Universal Robots PolyScope program: assembly_app.urp

Program assembly_app (installation=default directory=/home/ur/ursim-current/programs createdIn=5.17.1 lastSavedIn=5.17.1 robotSerialNumber=20195299999)
Calibrated DH parameters: a=[0, -0.6127, -0.57155, 0, 0, 0]; d=[0.1807, 0, 0, 0.17415, 0.11985, 0.11655]; alpha=[1.570796, 0, 0, 1.570796, -1.570796, 0]; deltaTheta=[0, 0, 0, 0, 0, 0]
InitVariablesNode
BeforeStart
  Script file /home/ur/ursim-current/programs/assemby_script_demo.script
    | # HMI input variables
    | approach = 100
    | contact_pose = p[-0.190, -0.610, 0.061, -0.00, 3.12, 0.04]
    | contact_force = 20
    | insertion_pose = p[-0.190, -0.610, 0.061, -0.00, 3.12, 0.04]
    | push_force = 30
    | step = 10
    | 
    | pick_pose = p[-0.189, -0.611, 0.240, -0.00, 3.11, 0.04]
    | threshold = 0.004
    | thread_running = False
    | 
    | # status variables
    | READY = 0
    | PICK = 1
    | APPROACH = 2
    | CONTACT = 3
    | SPIRAL = 4
    | INSERT = 5
    | ASSEMBLED = 6
    | status = READY
    | 
    | # thread functions for async movements
    | thread move_to_insert():
    |     movel(insertion_pose, v=0.02)
    |     thread_running = False
    | end
    | 
    | thread move_spiral():
    |     thread_running = False
    | end
    | 
    | # gripper functions
    | def grasp():
    | 
    | end
    | 
    | def release():
    | 
    | end
    | 
    | def pick():
    |     status = PICK
    |     sleep(2)
    | end
    | 
    | def assembly():
    |     # approach
    |     status = APPROACH
    |     sleep(2)
    | 
    |     # detect contact
    |     status = CONTACT
    |     sleep(2)
    | 
    |     # move spiral
    |     status = SPIRAL
    |     sleep(2)
    | 
    |     # insert
    |     status = INSERT
    |     sleep(2)
    | 
    |     # retract
    |     status = ASSEMBLED
    |     sleep(2)
    | end
    | 
    | # main function
    | def start_task():
    |     status = READY
    |     pick()
    |     assembly()
    | end
Robot Program (runOnlyOnce=false)
  URCap HMI (Robpod HMI URcap, Robpod Cloud) dataModel(robpod.hmi.selected=/home/ur/ursim-current/programs/assemby.hmi, robpod.hmi.stop.main.loop=true)
